// TIA Portal V21 export
// export: Created 2026-07-28T16:54:16.2567819Z, ExportSetting WithDefaults, DisplayName Totally Integrated Automation Portal, DisplayVersion V21, DisplayName SINAMICS Startdrive Advanced, DisplayVersion V21, DisplayName SINAMICS Startdrive G110M, G120, G120C, G120D, G120P, G115D, DisplayVersion V21, DisplayName SINAMICS Startdrive G130, G150, S120, S150, G200, G220, S200, S210, S220, Innomotics MVD, DisplayVersion V21, DisplayName STEP 7 Professional, DisplayVersion V21, DisplayName STEP 7 Safety, DisplayVersion V21, DisplayName Tech WebApplication, DisplayVersion V21, DisplayName WinCC Basic/Comfort/Advanced, DisplayVersion V21, DisplayName WinCC Professional, DisplayVersion V21, DisplayName WinCC Unified, DisplayVersion V21
TYPE "MotorPrincipal"
// Par principal/reserva com alternancia. Composicao em vez de campos duplicados:
//  os dois motores sao "MotorDados", e so o que e do PAR mora aqui.
//  Importar DEPOIS de MotorDados (o compilador exige o tipo referenciado ja existir).
// stored: IsFailsafeCompliant false
   STRUCT
      PRINCIPAL { S7_SetPoint := 'True'} : "MotorDados";
      RESERVA { S7_SetPoint := 'True'} : "MotorDados";   // --- comando do par (IHM) ---
      CMD_CHAVE_SELECAO_IHM : Byte;   // 0=alternancia 1=forca principal 2=forca reserva
      CMD_HABILITA_ALTERNANCIA : Bool;
      CMD_APLICAR_CADASTRO : Bool;   // copia SP_* do par pros dois motores
      CMD_RESET_FALHA_PAR : Bool;   // --- status do par ---
      STS_ATIVO_E_RESERVA : Bool;   // TRUE = o RESERVA esta assumindo o servico
      STS_PAR_DISPONIVEL : Bool;   // pelo menos um dos dois apto a partir
      STS_PAR_EM_FALHA : Bool;   // os dois indisponiveis
      STS_TEMPO_PARA_ALTERNAR : Real;   // [h] restante ate o proximo rodizio --- parametros do par ---
      SP_TEMPO_ROTATIVIDADE : Real;   // [h] intervalo de alternancia
      SP_TEMPO_SOBREPOSICAO : Real;   // [s] marcha simultanea na troca --- reserva ---
      RESERVA_BOOL_01 : Bool;
      RESERVA_INT_01 : Int;
      RESERVA_REAL_01 : Real;
   END_STRUCT;
END_TYPE
